// TwinCAT 3 PLC project stripper
// ProgramVersion: 3.1.4023.0
// libraries:
//   Tc2_DataExchange, * (Beckhoff Automation GmbH)
//   Tc2_Standard, * (Beckhoff Automation GmbH)
//   Tc2_System, * (Beckhoff Automation GmbH)
//   Tc3_Module, * (Beckhoff Automation GmbH)
// project tree:
//   FB/ FB_ReadAmsValue.TcPOU, FB_WriteAmsValue.TcPOU (not stored)
//   GVLs/ GVL.TcGVL, SUPVams.TcGVL (not stored)
//   / PlcTask.TcTTO
//   POUs/ MAIN.TcPOU, POU_readSupvData.TcPOU, POU_writeStripperToSupvData.TcPOU
// real-time tasks:
//   TASK PlcTask: cycle T#10ms, priority 20, ADS port 350

CONFIGURATION stripper
    RESOURCE PLC ON TwinCAT3
        TASK PlcTask(INTERVAL := T#10ms, PRIORITY := 20);
        PROGRAM MAIN WITH PlcTask : MAIN;
    END_RESOURCE
END_CONFIGURATION

// ---- GVLs/GVL.TcGVL
{attribute 'qualified_only'}
VAR_GLOBAL
	// setpoints
	PROD_RATE_SP					:	LREAL	:= 22.89;	// production rate
	L_STRIPPER_SP					:	LREAL	:= 50.0;	// stripper level
	L_SEPARATOR_SP					:	LREAL	:= 50.0;	// separator level
	L_REACTOR_SP					:	LREAL	:= 65.0;	// reactor level
	P_REACTOR_SP					:	LREAL;	// reactor pressure
	PCT_G_SP						:	LREAL;	// Mole percent G
	YA_SP							: 	LREAL;	// yA 
	YAC_SP							:	LREAL;	// yAC
	T_REACTOR_SP					:	LREAL;	// reactor temperature
	RECYC_VALVE_SP					:	LREAL;	// Recycle valve position
	STEAM_VALVE_SP					:	LREAL;	// Steam valve position
	L_AGITATOR_SP					:	LREAL;	// agitator setting		
	
	// Intermediate values
	Fp							:	LREAL; 		

	// actual production metrics
	COST						:	LREAL :=0.0;
	PctG						:	LREAL :=0.0;

	// process variables
	XMEAS						:	ARRAY[1..41] OF LREAL;
	XMEAS_TO_SUPV				:	ARRAY[1..10] OF LREAL; // 10,11-14,20,22,29-36
	
	XMV							:	ARRAY[1..12] OF LREAL;
	XMV_TO_SUPV					:	ARRAY[1..2] OF LREAL;  // 5,6,7
	
	// intermediate variables
	SEP_TEMP_SP					:	LREAL;	// separator temperaure setpoint
	RI							:	ARRAY[1..7] OF LREAL;	// ratio trimming outputs
	EADJ						:	LREAL;	// adjustment to production rate
	
	// shutdown indicator
	SD_FLAG						: 	BOOL	:= FALSE;

	// operating time
	OPTIME					:	LREAL := 0.0;		
END_VAR

// ---- POUs/MAIN.TcPOU
PROGRAM MAIN
VAR
END_VAR


POU_readSupvData();
POU_writeStripperToSupvData();

END_PROGRAM

// ---- POUs/POU_readSupvData.TcPOU
PROGRAM POU_readSupvData
VAR
	
	rUpdateRate : TIME := T#900MS;
	sNetId: T_AmsNetId := SUPVams.sNetId;	// '5.30.23.91.1.1';
	nPort: T_AmsPort := SUPVams.nPort; 		// 851

	nFpReadErrorId: UDINT;
	bFpReadError: BOOL;

	
	FB_ReadAmsValue_Fp: FB_ReadAmsValue;
	FB_ReadAmsValue_SPStripperLevel: FB_ReadAmsValue;
	FB_ReadAmsValue_SPPctG: FB_ReadAmsValue;
	
	bLStripReadError: BOOL;
	nFLStripReadErrorId: UDINT;
	bPctGReadError: BOOL;
	nPctGreadErrorId: UDINT;
END_VAR

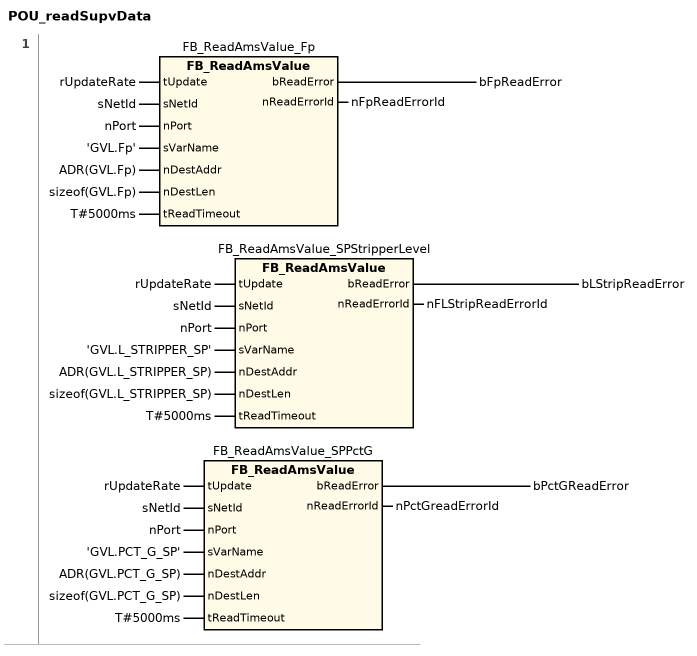
// NETWORK 1
FB_ReadAmsValue_Fp(
    tUpdate := rUpdateRate,
    sNetId := sNetId,
    nPort := nPort,
    sVarName := 'GVL.Fp',
    nDestAddr := ADR(GVL.Fp),
    nDestLen := sizeof(GVL.Fp),
    tReadTimeout := T#5000ms,
    nReadErrorId => nFpReadErrorId); // FB_ReadAmsValue
bFpReadError := FB_ReadAmsValue_Fp.bReadError;
FB_ReadAmsValue_SPStripperLevel(
    tUpdate := rUpdateRate,
    sNetId := sNetId,
    nPort := nPort,
    sVarName := 'GVL.L_STRIPPER_SP',
    nDestAddr := ADR(GVL.L_STRIPPER_SP),
    nDestLen := sizeof(GVL.L_STRIPPER_SP),
    tReadTimeout := T#5000ms,
    nReadErrorId => nFLStripReadErrorId); // FB_ReadAmsValue
bLStripReadError := FB_ReadAmsValue_SPStripperLevel.bReadError;
FB_ReadAmsValue_SPPctG(
    tUpdate := rUpdateRate,
    sNetId := sNetId,
    nPort := nPort,
    sVarName := 'GVL.PCT_G_SP',
    nDestAddr := ADR(GVL.PCT_G_SP),
    nDestLen := sizeof(GVL.PCT_G_SP),
    tReadTimeout := T#5000ms,
    nReadErrorId => nPctGreadErrorId); // FB_ReadAmsValue
bPctGReadError := FB_ReadAmsValue_SPPctG.bReadError;

END_PROGRAM

// ---- FB/FB_ReadAmsValue.TcPOU
FUNCTION_BLOCK FB_ReadAmsValue
VAR_INPUT
	tUpdate					:	TIME 				:=T#900MS;
	
	sNetId					:	T_AmsNetId			:='';
	nPort					:	T_AmsPort			:=851;
	sVarName				:	STRING(255)			:='';
	nDestAddr				:	PVOID;
	nDestLen				:	UDINT;
	tReadTimeout			:	TIME				:=T#2000MS;
	
END_VAR

VAR_OUTPUT
	bReadError		: BOOL := FALSE;
	nReadErrorId	: UDINT;
	
END_VAR

VAR
	
	ET_Read			: TIME := T#0MS;
	bReadEnable		: BOOL := FALSE;
	readBusy		: BOOL := FALSE;
	
	TON_Read		: TON;
	fb_reader	: FB_ReadAdsSymByName;
END_VAR

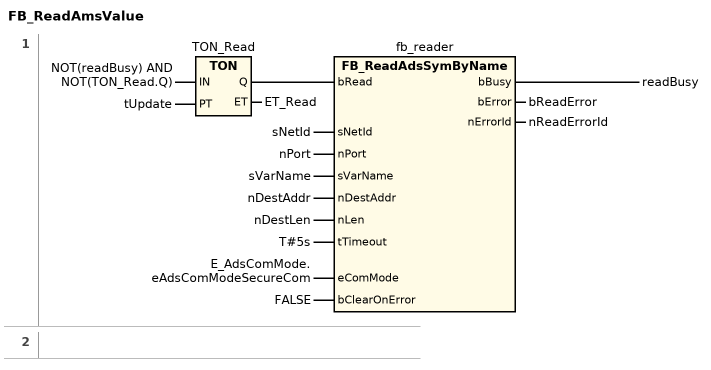
// NETWORK 1
TON_Read(IN := NOT(readBusy) AND NOT(TON_Read.Q), PT := tUpdate, ET => ET_Read); // TON
fb_reader(
    bRead := TON_Read.Q,
    sNetId := sNetId,
    nPort := nPort,
    sVarName := sVarName,
    nDestAddr := nDestAddr,
    nLen := nDestLen,
    tTimeout := T#5s,
    eComMode := E_AdsComMode.eAdsComModeSecureCom,
    bClearOnError := FALSE,
    bError => bReadError,
    nErrorId => nReadErrorId); // FB_ReadAdsSymByName
readBusy := fb_reader.bBusy;

// NETWORK 2

END_FUNCTION_BLOCK

// ---- POUs/POU_writeStripperToSupvData.TcPOU
PROGRAM POU_writeStripperToSupvData
VAR
	rUpdateRate : TIME := T#900MS;	
	sNetId: T_AmsNetId := SUPVams.sNetId;	// '5.30.23.91.1.1';
	nPort: T_AmsPort := SUPVams.nPort; 		// 851	

	FB_WriteAmsValue_XMEAS: FB_WriteAmsValue;
	FB_WriteAmsValue_XMV: FB_WriteAmsValue;
	nXMEASWriteErrorId: UDINT;
	bXMEASWriteError: BOOL;
	bXMVWriteError: BOOL;
	nXMVWriteErrorId: UDINT;
	
	FB_WriteAmsValue_EADJ: FB_WriteAmsValue;
	nEADJWriteErrorId: UDINT;
	bEADJWriteError: BOOL;
	FB_WriteAmsValue_PctG: FB_WriteAmsValue;
	bPctGWriteError: BOOL;
END_VAR

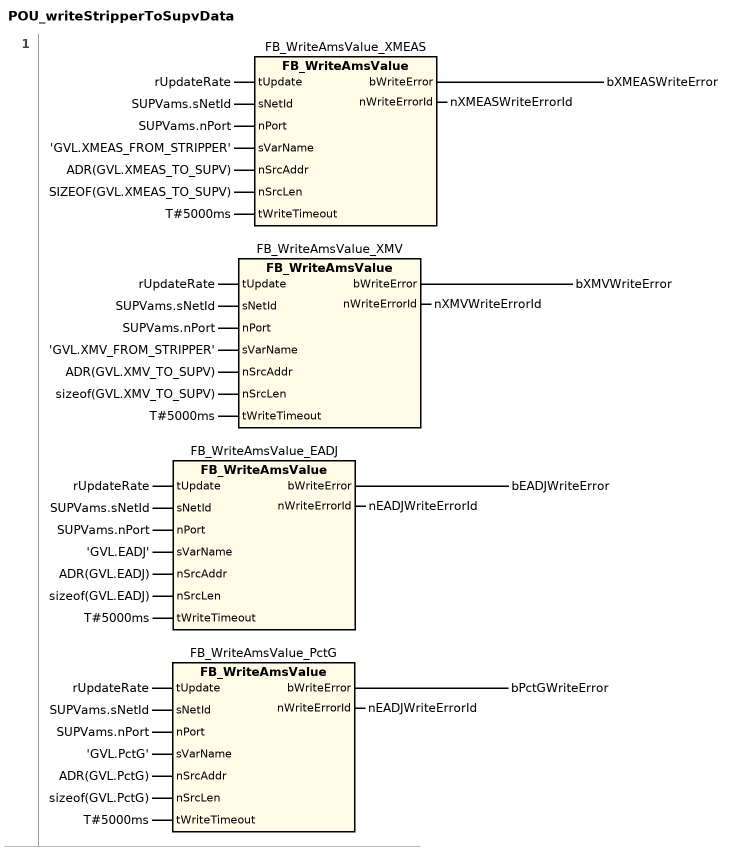
// NETWORK 1
FB_WriteAmsValue_XMEAS(
    tUpdate := rUpdateRate,
    sNetId := SUPVams.sNetId,
    nPort := SUPVams.nPort,
    sVarName := 'GVL.XMEAS_FROM_STRIPPER',
    nSrcAddr := ADR(GVL.XMEAS_TO_SUPV),
    nSrcLen := SIZEOF(GVL.XMEAS_TO_SUPV),
    tWriteTimeout := T#5000ms,
    nWriteErrorId => nXMEASWriteErrorId); // FB_WriteAmsValue
bXMEASWriteError := FB_WriteAmsValue_XMEAS.bWriteError;
FB_WriteAmsValue_XMV(
    tUpdate := rUpdateRate,
    sNetId := SUPVams.sNetId,
    nPort := SUPVams.nPort,
    sVarName := 'GVL.XMV_FROM_STRIPPER',
    nSrcAddr := ADR(GVL.XMV_TO_SUPV),
    nSrcLen := sizeof(GVL.XMV_TO_SUPV),
    tWriteTimeout := T#5000ms,
    nWriteErrorId => nXMVWriteErrorId); // FB_WriteAmsValue
bXMVWriteError := FB_WriteAmsValue_XMV.bWriteError;
FB_WriteAmsValue_EADJ(
    tUpdate := rUpdateRate,
    sNetId := SUPVams.sNetId,
    nPort := SUPVams.nPort,
    sVarName := 'GVL.EADJ',
    nSrcAddr := ADR(GVL.EADJ),
    nSrcLen := sizeof(GVL.EADJ),
    tWriteTimeout := T#5000ms,
    nWriteErrorId => nEADJWriteErrorId); // FB_WriteAmsValue
bEADJWriteError := FB_WriteAmsValue_EADJ.bWriteError;
FB_WriteAmsValue_PctG(
    tUpdate := rUpdateRate,
    sNetId := SUPVams.sNetId,
    nPort := SUPVams.nPort,
    sVarName := 'GVL.PctG',
    nSrcAddr := ADR(GVL.PctG),
    nSrcLen := sizeof(GVL.PctG),
    tWriteTimeout := T#5000ms,
    nWriteErrorId => nEADJWriteErrorId); // FB_WriteAmsValue
bPctGWriteError := FB_WriteAmsValue_PctG.bWriteError;

END_PROGRAM
